FUNCTION_BLOCK TEST_PRINT (* Test Java println() function in ST algorithm *)
  (* Standard: 61499-2 *)
  (* Version 0.0, 2002-12-17, JHC, Rockwell Automation *)
  (* Compiler header: package fb.rt.test; *)
  (* Compiler Java IBM Jikes 1.06 *)
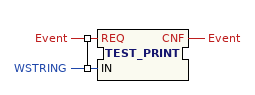
  EVENT_INPUT
    REQ WITH IN; (* Normal Execution Request *)
  END_EVENT
  EVENT_OUTPUT
    CNF; (* Execution Confirmation *)
  END_EVENT
  VAR_INPUT
    IN : WSTRING; (* Data to print *)
  END_VAR
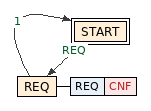
  EC_STATES
    START; (* Initial State *)
    REQ : REQ -> CNF; (* Normal execution *)
  END_STATES
  EC_TRANSITIONS
    START TO REQ := REQ;
    REQ TO START := 1;
  END_TRANSITIONS
  ALGORITHM REQ IN ST: (* Normally executed algorithm *)
System.out.println(IN);
  END_ALGORITHM
END_FUNCTION_BLOCK
